// TIA Portal V18 export
TYPE "UDT_AHUEqpDataType"
// stored: IsFailsafeCompliant false
   STRUCT
      cFan : Array[1..3] of Byte;   // 0-wout ctrl/1 - ProxiAdaptation/
      cExtractDumper : Array[1..3] of Byte;   // 0-wout ctrl/1 - ProxiAdaptation/
      cMixingDumper : Array[1..3] of Byte;   // 0-wout ctrl/1 - ProxiAdaptation/
      cHeater : Array[1..3] of Byte;   // 0-wout ctrl/1 - ProxiAdaptation/
      cCooler : Array[1..3] of Byte;   // 0-wout ctrl/1 - ProxiAdaptation/
      cWHU : Array[1..3] of Byte;   // 0-wout ctrl/1 - ProxiAdaptation/
   END_STRUCT;
END_TYPE
